INTERFACE I_AxisControl EXTENDS __SYSTEM.IQueryInterface

PROPERTY PUBLIC Acceleration : mc_lreal
GET
END_GET
SET
END_SET
END_PROPERTY

PROPERTY BufferMode : MC_BufferMode
GET
END_GET
SET
END_SET
END_PROPERTY

PROPERTY PUBLIC Deceleration : mc_lreal
GET
END_GET
SET
END_SET
END_PROPERTY

METHOD DisableAxis : HRESULT
VAR_INPUT
END_VAR
END_METHOD

METHOD EnableAxis : HRESULT
VAR_INPUT
END_VAR
END_METHOD

METHOD HaltAxis : HRESULT
VAR_INPUT
END_VAR
END_METHOD

PROPERTY PUBLIC Jerk : mc_lreal
GET
END_GET
SET
END_SET
END_PROPERTY

METHOD MoveToPosition : HRESULT
VAR_INPUT
	Position : MC_LREAL;
	Velocity : MC_LREAL;
END_VAR
END_METHOD

METHOD Reset : HRESULT
VAR_INPUT
END_VAR
END_METHOD

END_INTERFACE

(* stored: Version 1.1.0.1
   Itf I_AxisControl: Id {67ee2d44-07ee-4a7f-8cf0-2ba796d7942a}
   Property Acceleration: Id {6aa38efd-5aab-4e71-a9b5-4601e763ad20}
   Get Get: Id {2772526e-ce15-4b61-8310-c1fa3f5374d7}
   Set Set: Id {c4d5c93b-6bb9-430e-bfdc-58ca88aea98e}
   Property BufferMode: Id {8a09ec3d-50cb-4ca8-b8b1-13388b194d0f}
   Get Get: Id {25d07f96-89ca-4e5a-9a52-920a8faf68e1}
   Set Set: Id {16124384-c0ca-494a-b3ee-94016c9eddae}
   Property Deceleration: Id {f4545876-9890-47b0-a794-487261b1a669}
   Get Get: Id {61cc8aaf-c6b0-4c2f-b29e-5a00fbd2b6ef}
   Set Set: Id {cbee0af5-61c7-45cc-aee3-6fc8bb0b9c3f}
   Method DisableAxis: Id {78e4be45-9441-4dfd-be50-a8de43882816}
   Method EnableAxis: Id {dc495f2e-73cd-4872-9d3b-75cfe930dc9c}
   Method HaltAxis: Id {94883e86-e022-461f-9256-2ce498881fb1}
   Property Jerk: Id {0df40572-608e-4996-8cc9-9fa0ad407b16}
   Get Get: Id {0bff625d-12a6-41b9-9a30-2b50870310c3}
   Set Set: Id {7c979efc-b6ea-40bb-b0fd-ca613f140f10}
   Method MoveToPosition: Id {c5eac34c-4010-4d8b-8622-96313c7f08cf}
   Method Reset: Id {fe6c826c-85ca-40eb-8eb2-4dba05c9813a} *)
